(* CoDeSys 2.3 export: BUTTONTRIGGEREDTIMEDONOFF.EXP *)

(* POU Components/OnOff/ButtonTriggeredTimedOnOff, ST *)
FUNCTION_BLOCK ButtonTriggeredTimedOnOff
VAR_INPUT
	input:BOOL;
	timeSetup:INT;
END_VAR
VAR_OUTPUT
	output:BOOL;
END_VAR
VAR
	Button:Button;
	TimedOnOff:TimedOnOff;
	state:BOOL;
END_VAR
button(input:=input);
timedOnOff(timeSetup:=timeSetup, input:= button.fallingEdge, permanent:= button.longPressed, output=>output);
state:=timedOnOff.state;
END_FUNCTION_BLOCK
